TYPE ST_MAIN_MODULE :
STRUCT

	TEMP_CONTROLLER:ST_TEMP_CONTROLLER;  // 구조가 변결 될 수  있음
	LINE_HEATER:ARRAY[1..8] OF ST_TEMP_CONTROLLER;// 구조가 변결 될 수  있음
	BATH_TEMP:ARRAY[1..3]OF ST_TEMP_CONTROLLER;
	THROTTLE_VALVE:ST_THROTTLE_VALVE;// 구조가 변결 될 수  있음
	ROTATION_MOTOR:ST_ROTATION_MOTOR; // jhkang_251112 추가됨
	UTILITY:ST_UTILITY;
END_STRUCT
END_TYPE

(* stored: Version 1.1.0.1, ProductVersion 3.1.4024.12
   DUT ST_MAIN_MODULE: Id {25f5eb89-ca03-4585-b681-bf62172c38ca} *)
